
// ===== library: MasterCopy "Pulzer" =====

FUNCTION "Pulzer" : Void   // FC2, LAD
{ S7_Optimized_Access := 'FALSE' }
VERSION : 0.1
   VAR_INPUT
      T1 : Timer;
      T2 : Timer;
      Thigh : S5Time;
      Tdown : S5Time;
   END_VAR
   VAR_OUTPUT
      Q : Bool;
   END_VAR
   VAR_TEMP   // added for the SCL form of the ladder/FBD networks
      _w1 : Bool;
      _s5time1 : S5Time;
   END_VAR
BEGIN

REGION Network 1
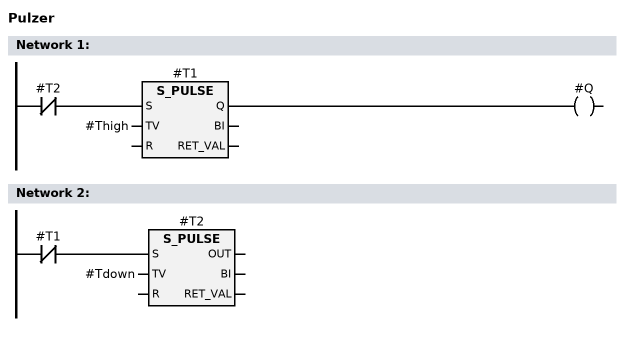
   RUNG wire#powerrail
      I_Contact( #T2 )
      S_PULSE(T_NO := #T1, TV := #Thigh, R :=, BI =>, RET_VAL =>)
      Coil( #Q )
   END_RUNG
   // the same network as SCL:
   #_s5time1 := S_PULSE(T_NO := #T1, S := NOT #T2, TV := #Thigh, Q => #_w1);
   #Q := #_w1;
END_REGION

REGION Network 2
   RUNG wire#powerrail
      I_Contact( #T1 )
      S_PULSE(T_NO := #T2, TV := #Tdown, R :=, BI =>, RET_VAL =>)
   END_RUNG
   // the same network as SCL:
   #_s5time1 := S_PULSE(T_NO := #T2, S := NOT #T1, TV := #Tdown);
END_REGION
END_FUNCTION

// ===== library: MasterCopy "Pallet dispenser" =====

FUNCTION_BLOCK "Pallet dispenser"   // FB4, LAD
{ S7_Optimized_Access := 'FALSE' }
VERSION : 0.1
   VAR_INPUT
      DOWN_accident : Bool;
      Dispenser_is_down : Bool;
      Dispenser_in_middle : Bool;
      Dispenser_is_up : Bool;
      UP_accident : Bool;
      Circuit_breaker : Bool;
      Arms_are_open : Bool;
      Arms_are_close : Bool;
      Pallet_under_dispenser : Bool;
      Automatic_mode : Bool;
      Power_circuit_OK : Bool;
      Pneumatic_OK : Bool;
      Sensor_before_dispenser : Bool;
      Button_Open_door : Bool;
      Sensor_door_are_open : Bool;
      Button_Door_are_close : Bool;
      OP_up : Bool;
      OP_down : Bool;
      OP_Airs_move : Bool;
      Pallet_transfare : Bool;
      Button_RESET : Bool;
      "Časovač 1" : Timer;
      "Časovač 2" : Timer;
      "Časovač 3" : Timer;
      "Časovač 4" : Timer;
      "Časovač 5" : Timer;
   END_VAR
   VAR_OUTPUT
      Let_go_UP : Bool;
      Let_go_DOWN : Bool;
      Break : Bool;
      Let_arms_close : Bool;
      Let_arms_open : Bool;
      Let_open_door : Bool;
      Led_door_are_open : Bool;
   END_VAR
   VAR
      Paleta_polozena : Bool;
      Stop_v_rucnim : Bool;
      Hrana_stop_v_rucnim : Bool;
      Pozadavek_otevreni_dveri : Bool;
      Door_opened : Bool;
      Arms_are_close_pozition : Bool;
   END_VAR
   VAR_TEMP   // added for the SCL form of the ladder/FBD networks
      _s5time1 : S5Time;
      _w1 : Bool;
   END_VAR
BEGIN

REGION Network 1
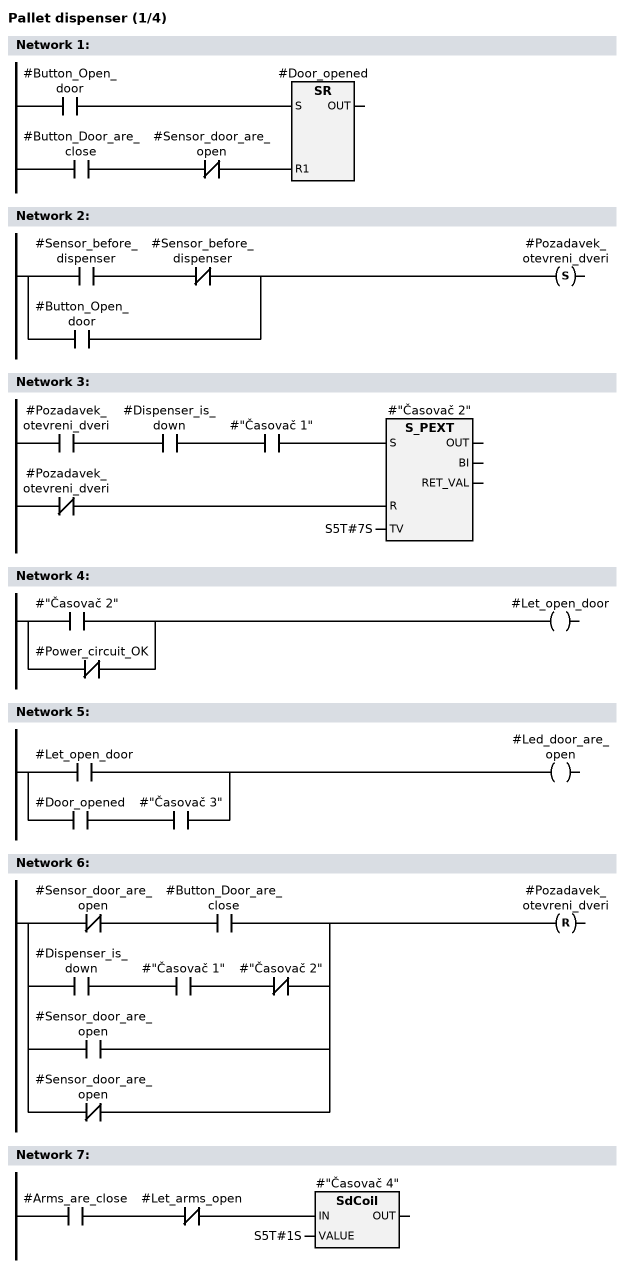
   RUNG wire#powerrail
      Contact( #Button_Open_door )
      S_SR(operand := #Door_opened, r1 := wire#w1)
   END_RUNG
   RUNG wire#powerrail
      Contact( #Button_Door_are_close )
      I_Contact( #Sensor_door_are_open )
   END_RUNG wire#w1
   // the same network as SCL:
   IF #Button_Open_door THEN
       #Door_opened := TRUE;   // SR flip-flop
   END_IF;
   IF #Button_Door_are_close AND NOT #Sensor_door_are_open THEN #Door_opened := FALSE; END_IF;
END_REGION

REGION Network 2
   RUNG wire#powerrail
      Contact( #Sensor_before_dispenser )
      I_Contact( #Sensor_before_dispenser )
      wire#w1
      S_Coil( #Pozadavek_otevreni_dveri )
   END_RUNG
   RUNG wire#powerrail
      Contact( #Button_Open_door )
   END_RUNG wire#w1
   // the same network as SCL:
   IF (#Sensor_before_dispenser AND NOT #Sensor_before_dispenser) OR #Button_Open_door THEN
       #Pozadavek_otevreni_dveri := TRUE;
   END_IF;
END_REGION

REGION Network 3
   RUNG wire#powerrail
      Contact( #Pozadavek_otevreni_dveri )
      Contact( #Dispenser_is_down )
      Contact( #"Časovač 1" )
      S_PEXT(T_NO := #"Časovač 2", R := wire#w1, TV := S5T#7S, BI =>, RET_VAL =>)
   END_RUNG
   RUNG wire#powerrail
      I_Contact( #Pozadavek_otevreni_dveri )
   END_RUNG wire#w1
   // the same network as SCL:
   #_s5time1 := S_PEXT(T_NO := #"Časovač 2",
                       S := #Pozadavek_otevreni_dveri AND #Dispenser_is_down AND #"Časovač 1",
                       R := NOT #Pozadavek_otevreni_dveri,
                       TV := S5T#7S);
END_REGION

REGION Network 4
   RUNG wire#powerrail
      Contact( #"Časovač 2" )
      wire#w1
      Coil( #Let_open_door )
   END_RUNG
   RUNG wire#powerrail
      I_Contact( #Power_circuit_OK )
   END_RUNG wire#w1
   // the same network as SCL:
   #Let_open_door := #"Časovač 2" OR NOT #Power_circuit_OK;
END_REGION

REGION Network 5
   RUNG wire#powerrail
      Contact( #Let_open_door )
      wire#w1
      Coil( #Led_door_are_open )
   END_RUNG
   RUNG wire#powerrail
      Contact( #Door_opened )
      Contact( #"Časovač 3" )
   END_RUNG wire#w1
   // the same network as SCL:
   #Led_door_are_open := #Let_open_door OR (#Door_opened AND #"Časovač 3");
END_REGION

REGION Network 6
   RUNG wire#powerrail
      I_Contact( #Sensor_door_are_open )
      Contact( #Button_Door_are_close )
      wire#w1
      R_Coil( #Pozadavek_otevreni_dveri )
   END_RUNG
   RUNG wire#powerrail
      Contact( #Dispenser_is_down )
      Contact( #"Časovač 1" )
      I_Contact( #"Časovač 2" )
   END_RUNG wire#w1
   RUNG wire#powerrail
      Contact( #Sensor_door_are_open )
   END_RUNG wire#w1
   RUNG wire#powerrail
      I_Contact( #Sensor_door_are_open )
   END_RUNG wire#w1
   // the same network as SCL:
   IF (NOT #Sensor_door_are_open AND #Button_Door_are_close) OR (#Dispenser_is_down AND #"Časovač 1" AND NOT #"Časovač 2") OR #Sensor_door_are_open OR NOT #Sensor_door_are_open THEN
       #Pozadavek_otevreni_dveri := FALSE;
   END_IF;
END_REGION

REGION Network 7
   // no SCL statement known for SdCoil: written as a call
   SdCoil(in := #Arms_are_close AND NOT #Let_arms_open, value := S5T#1S, operand := #"Časovač 4");
END_REGION

REGION Network 8
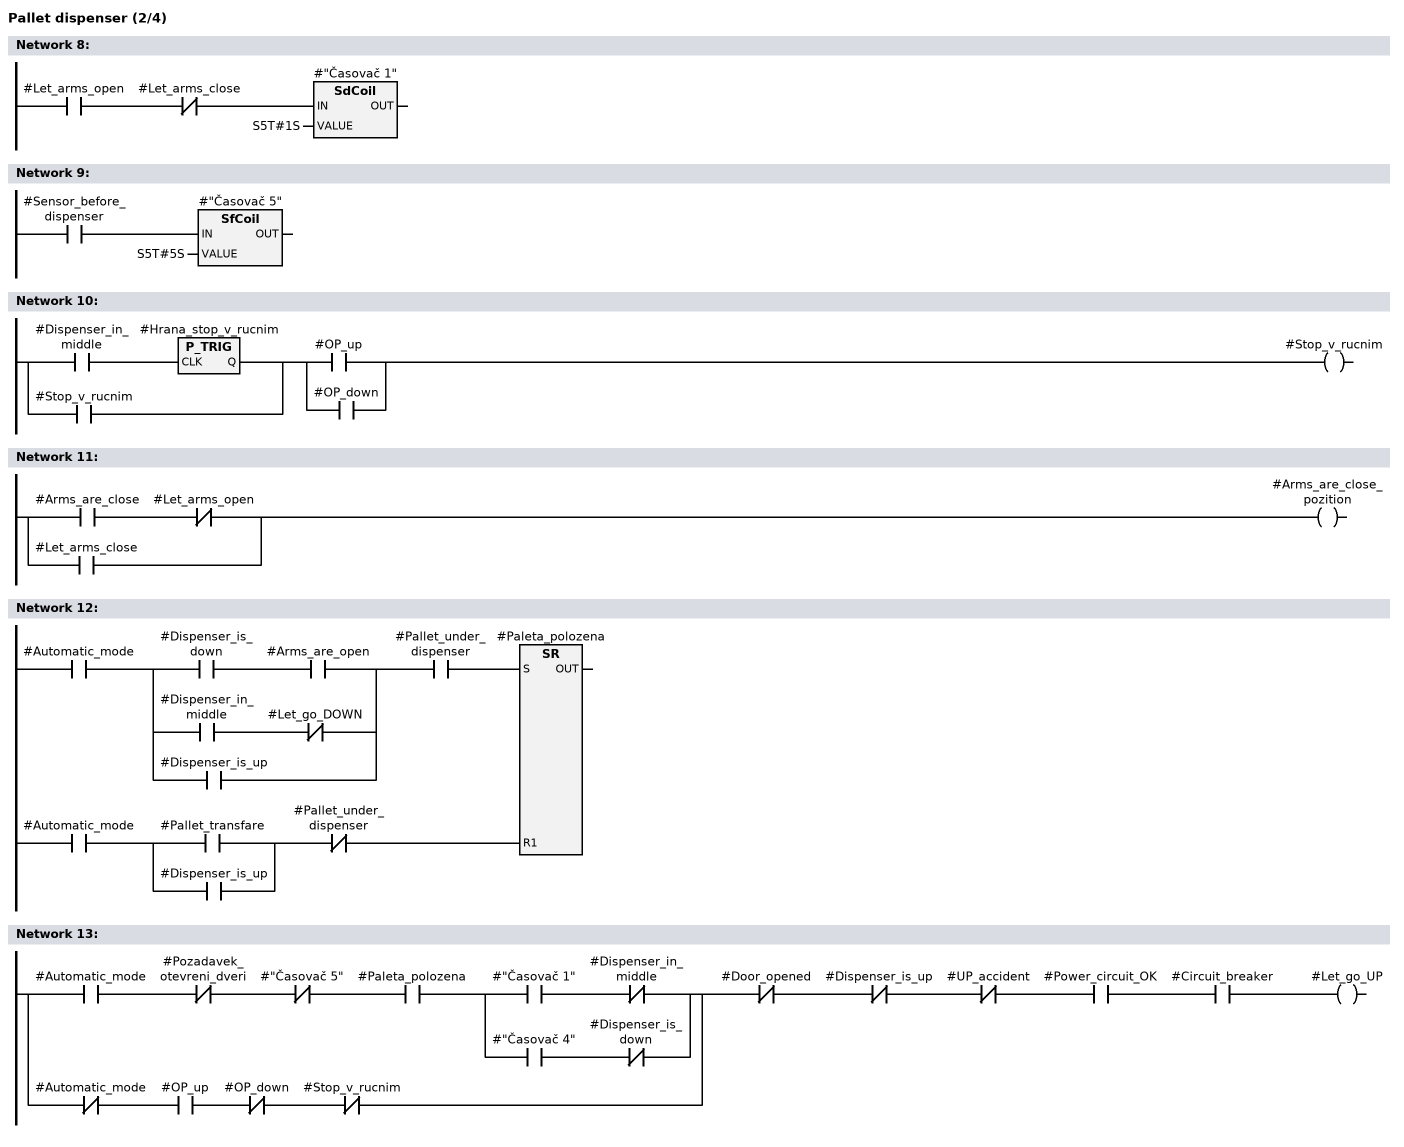
   // no SCL statement known for SdCoil: written as a call
   SdCoil(in := #Let_arms_open AND NOT #Let_arms_close, value := S5T#1S, operand := #"Časovač 1");
END_REGION

REGION Network 9
   // no SCL statement known for SfCoil: written as a call
   SfCoil(in := #Sensor_before_dispenser, value := S5T#5S, operand := #"Časovač 5");
END_REGION

REGION Network 10
   RUNG wire#powerrail
      Contact( #Dispenser_in_middle )
      P_Trig( #Hrana_stop_v_rucnim )
      wire#w1
      Contact( #OP_up )
      wire#w2
      Coil( #Stop_v_rucnim )
   END_RUNG
   RUNG wire#powerrail
      Contact( #Stop_v_rucnim )
   END_RUNG wire#w1
   RUNG wire#w1
      Contact( #OP_down )
   END_RUNG wire#w2
   // the same network as SCL:
   #_w1 := #Dispenser_in_middle AND NOT #Hrana_stop_v_rucnim;   // rising edge
   #Hrana_stop_v_rucnim := #Dispenser_in_middle;
   #Stop_v_rucnim := (#_w1 OR #Stop_v_rucnim) AND (#OP_up OR #OP_down);
END_REGION

REGION Network 11
   RUNG wire#powerrail
      Contact( #Arms_are_close )
      I_Contact( #Let_arms_open )
      wire#w1
      Coil( #Arms_are_close_pozition )
   END_RUNG
   RUNG wire#powerrail
      Contact( #Let_arms_close )
   END_RUNG wire#w1
   // the same network as SCL:
   #Arms_are_close_pozition := (#Arms_are_close AND NOT #Let_arms_open) OR #Let_arms_close;
END_REGION

REGION Network 12
   RUNG wire#powerrail
      Contact( #Automatic_mode )
      wire#w1
      Contact( #Dispenser_is_down )
      Contact( #Arms_are_open )
      wire#w2
      Contact( #Pallet_under_dispenser )
      S_SR(operand := #Paleta_polozena, r1 := wire#w5)
   END_RUNG
   RUNG wire#w1
      Contact( #Dispenser_in_middle )
      I_Contact( #Let_go_DOWN )
   END_RUNG wire#w2
   RUNG wire#w1
      Contact( #Dispenser_is_up )
   END_RUNG wire#w2
   RUNG wire#powerrail
      Contact( #Automatic_mode )
      wire#w3
      Contact( #Pallet_transfare )
      wire#w4
      I_Contact( #Pallet_under_dispenser )
   END_RUNG wire#w5
   RUNG wire#w3
      Contact( #Dispenser_is_up )
   END_RUNG wire#w4
   // the same network as SCL:
   IF #Automatic_mode AND ((#Dispenser_is_down AND #Arms_are_open) OR (#Dispenser_in_middle AND NOT #Let_go_DOWN) OR #Dispenser_is_up) AND #Pallet_under_dispenser THEN
       #Paleta_polozena := TRUE;   // SR flip-flop
   END_IF;
   IF #Automatic_mode AND (#Pallet_transfare OR #Dispenser_is_up) AND NOT #Pallet_under_dispenser THEN
       #Paleta_polozena := FALSE;
   END_IF;
END_REGION

REGION Network 13
   RUNG wire#powerrail
      Contact( #Automatic_mode )
      I_Contact( #Pozadavek_otevreni_dveri )
      I_Contact( #"Časovač 5" )
      Contact( #Paleta_polozena )
      wire#w1
      Contact( #"Časovač 1" )
      I_Contact( #Dispenser_in_middle )
      wire#w2
      I_Contact( #Door_opened )
      I_Contact( #Dispenser_is_up )
      I_Contact( #UP_accident )
      Contact( #Power_circuit_OK )
      Contact( #Circuit_breaker )
      Coil( #Let_go_UP )
   END_RUNG
   RUNG wire#w1
      Contact( #"Časovač 4" )
      I_Contact( #Dispenser_is_down )
   END_RUNG wire#w2
   RUNG wire#powerrail
      I_Contact( #Automatic_mode )
      Contact( #OP_up )
      I_Contact( #OP_down )
      I_Contact( #Stop_v_rucnim )
   END_RUNG wire#w2
   // the same network as SCL:
   #Let_go_UP := ((#Automatic_mode AND NOT #Pozadavek_otevreni_dveri AND NOT #"Časovač 5" AND #Paleta_polozena AND ((#"Časovač 1" AND NOT #Dispenser_in_middle) OR (#"Časovač 4" AND NOT #Dispenser_is_down))) OR (NOT #Automatic_mode AND #OP_up AND NOT #OP_down AND NOT #Stop_v_rucnim)) AND NOT #Door_opened AND NOT #Dispenser_is_up AND NOT #UP_accident AND #Power_circuit_OK AND #Circuit_breaker;
END_REGION

REGION Network 14
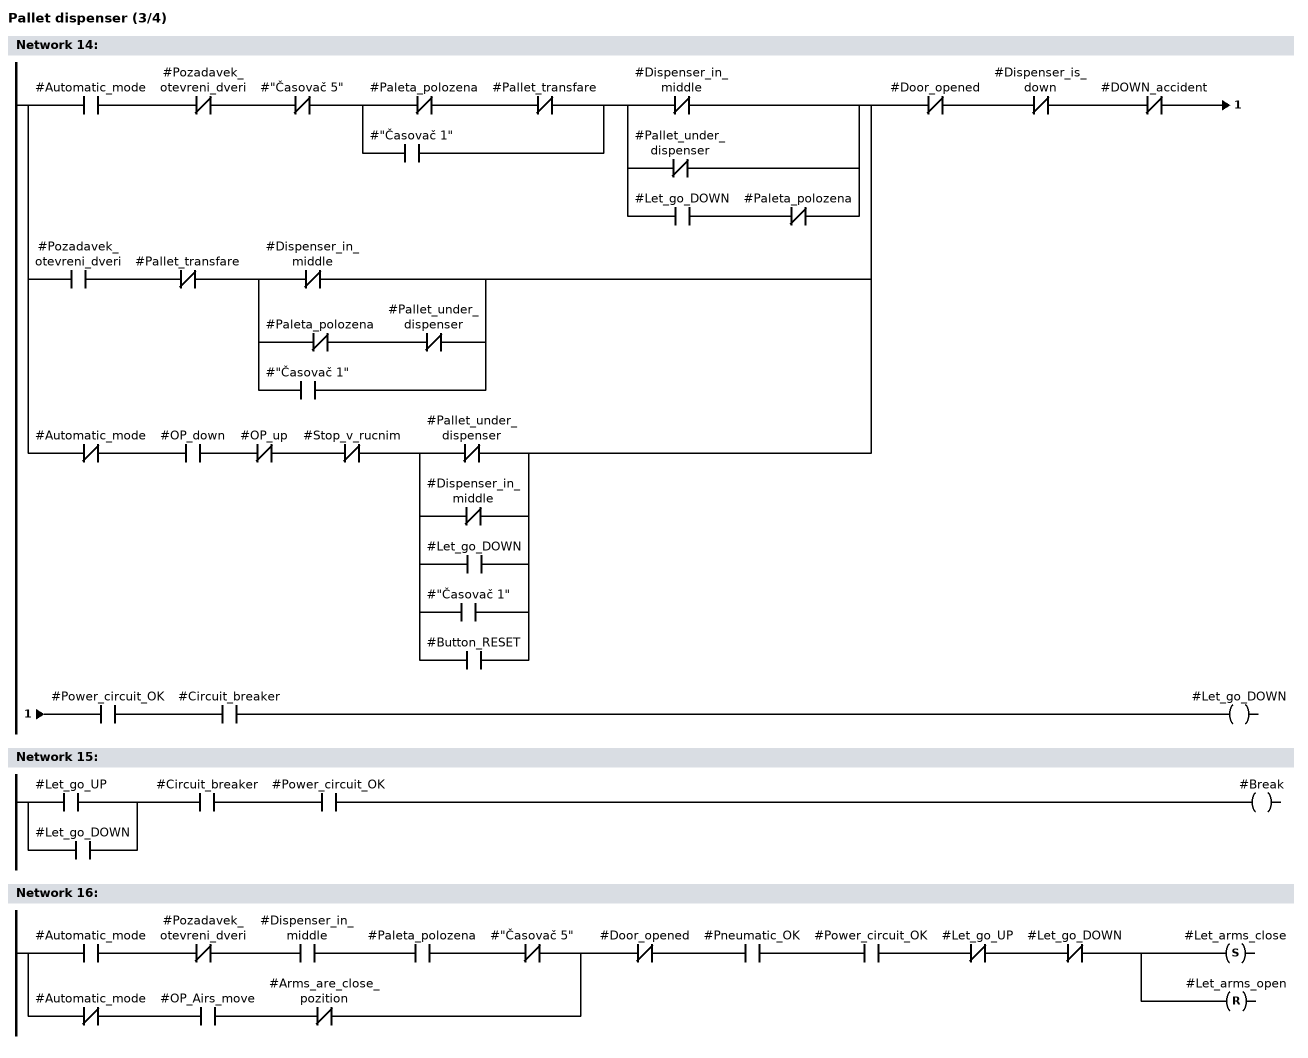
   RUNG wire#powerrail
      Contact( #Automatic_mode )
      I_Contact( #Pozadavek_otevreni_dveri )
      I_Contact( #"Časovač 5" )
      wire#w1
      I_Contact( #Paleta_polozena )
      I_Contact( #Pallet_transfare )
      wire#w2
      I_Contact( #Dispenser_in_middle )
      wire#w3
      I_Contact( #Door_opened )
      I_Contact( #Dispenser_is_down )
      I_Contact( #DOWN_accident )
      Contact( #Power_circuit_OK )
      Contact( #Circuit_breaker )
      Coil( #Let_go_DOWN )
   END_RUNG
   RUNG wire#w1
      Contact( #"Časovač 1" )
   END_RUNG wire#w2
   RUNG wire#w2
      I_Contact( #Pallet_under_dispenser )
   END_RUNG wire#w3
   RUNG wire#w2
      Contact( #Let_go_DOWN )
      I_Contact( #Paleta_polozena )
   END_RUNG wire#w3
   RUNG wire#powerrail
      Contact( #Pozadavek_otevreni_dveri )
      I_Contact( #Pallet_transfare )
      wire#w4
      I_Contact( #Dispenser_in_middle )
   END_RUNG wire#w3
   RUNG wire#w4
      I_Contact( #Paleta_polozena )
      I_Contact( #Pallet_under_dispenser )
   END_RUNG wire#w3
   RUNG wire#w4
      Contact( #"Časovač 1" )
   END_RUNG wire#w3
   RUNG wire#powerrail
      I_Contact( #Automatic_mode )
      Contact( #OP_down )
      I_Contact( #OP_up )
      I_Contact( #Stop_v_rucnim )
      wire#w5
      I_Contact( #Pallet_under_dispenser )
   END_RUNG wire#w3
   RUNG wire#w5
      I_Contact( #Dispenser_in_middle )
   END_RUNG wire#w3
   RUNG wire#w5
      Contact( #Let_go_DOWN )
   END_RUNG wire#w3
   RUNG wire#w5
      Contact( #"Časovač 1" )
   END_RUNG wire#w3
   RUNG wire#w5
      Contact( #Button_RESET )
   END_RUNG wire#w3
   // the same network as SCL:
   #Let_go_DOWN := ((#Automatic_mode AND NOT #Pozadavek_otevreni_dveri AND NOT #"Časovač 5" AND ((NOT #Paleta_polozena AND NOT #Pallet_transfare) OR #"Časovač 1") AND (NOT #Dispenser_in_middle OR NOT #Pallet_under_dispenser OR (#Let_go_DOWN AND NOT #Paleta_polozena))) OR (#Pozadavek_otevreni_dveri AND NOT #Pallet_transfare AND (NOT #Dispenser_in_middle OR (NOT #Paleta_polozena AND NOT #Pallet_under_dispenser) OR #"Časovač 1")) OR (NOT #Automatic_mode AND #OP_down AND NOT #OP_up AND NOT #Stop_v_rucnim AND (NOT #Pallet_under_dispenser OR NOT #Dispenser_in_middle OR #Let_go_DOWN OR #"Časovač 1" OR #Button_RESET))) AND NOT #Door_opened AND NOT #Dispenser_is_down AND NOT #DOWN_accident AND #Power_circuit_OK AND #Circuit_breaker;
END_REGION

REGION Network 15
   RUNG wire#powerrail
      Contact( #Let_go_UP )
      wire#w1
      Contact( #Circuit_breaker )
      Contact( #Power_circuit_OK )
      Coil( #Break )
   END_RUNG
   RUNG wire#powerrail
      Contact( #Let_go_DOWN )
   END_RUNG wire#w1
   // the same network as SCL:
   #Break := (#Let_go_UP OR #Let_go_DOWN) AND #Circuit_breaker AND #Power_circuit_OK;
END_REGION

REGION Network 16
   RUNG wire#powerrail
      Contact( #Automatic_mode )
      I_Contact( #Pozadavek_otevreni_dveri )
      Contact( #Dispenser_in_middle )
      Contact( #Paleta_polozena )
      I_Contact( #"Časovač 5" )
      wire#w1
      I_Contact( #Door_opened )
      Contact( #Pneumatic_OK )
      Contact( #Power_circuit_OK )
      I_Contact( #Let_go_UP )
      I_Contact( #Let_go_DOWN )
      wire#w2
      S_Coil( #Let_arms_close )
   END_RUNG
   RUNG wire#powerrail
      I_Contact( #Automatic_mode )
      Contact( #OP_Airs_move )
      I_Contact( #Arms_are_close_pozition )
   END_RUNG wire#w1
   RUNG wire#w2
      R_Coil( #Let_arms_open )
   END_RUNG
   // the same network as SCL:
   IF ((#Automatic_mode AND NOT #Pozadavek_otevreni_dveri AND #Dispenser_in_middle AND #Paleta_polozena AND NOT #"Časovač 5") OR (NOT #Automatic_mode AND #OP_Airs_move AND NOT #Arms_are_close_pozition)) AND NOT #Door_opened AND #Pneumatic_OK AND #Power_circuit_OK AND NOT #Let_go_UP AND NOT #Let_go_DOWN THEN
       #Let_arms_close := TRUE;
       #Let_arms_open := FALSE;
   END_IF;
END_REGION

REGION Network 17
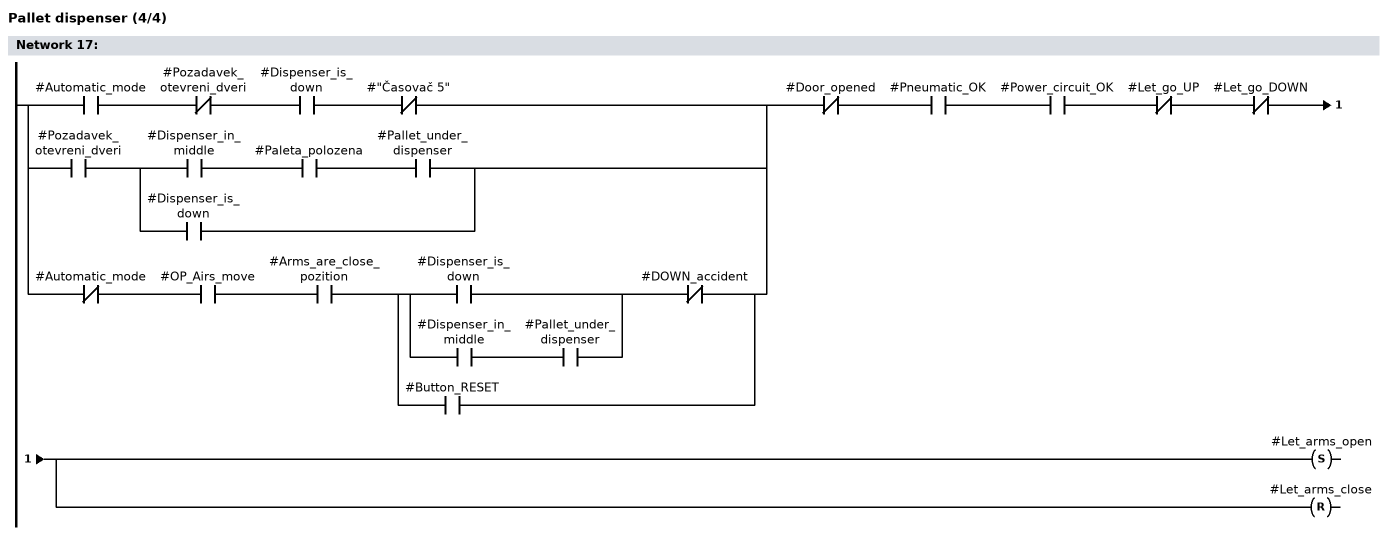
   RUNG wire#powerrail
      Contact( #Automatic_mode )
      I_Contact( #Pozadavek_otevreni_dveri )
      Contact( #Dispenser_is_down )
      I_Contact( #"Časovač 5" )
      wire#w1
      I_Contact( #Door_opened )
      Contact( #Pneumatic_OK )
      Contact( #Power_circuit_OK )
      I_Contact( #Let_go_UP )
      I_Contact( #Let_go_DOWN )
      wire#w5
      S_Coil( #Let_arms_open )
   END_RUNG
   RUNG wire#powerrail
      Contact( #Pozadavek_otevreni_dveri )
      wire#w2
      Contact( #Dispenser_in_middle )
      Contact( #Paleta_polozena )
      Contact( #Pallet_under_dispenser )
   END_RUNG wire#w1
   RUNG wire#w2
      Contact( #Dispenser_is_down )
   END_RUNG wire#w1
   RUNG wire#powerrail
      I_Contact( #Automatic_mode )
      Contact( #OP_Airs_move )
      Contact( #Arms_are_close_pozition )
      wire#w3
      Contact( #Dispenser_is_down )
      wire#w4
      I_Contact( #DOWN_accident )
   END_RUNG wire#w1
   RUNG wire#w3
      Contact( #Dispenser_in_middle )
      Contact( #Pallet_under_dispenser )
   END_RUNG wire#w4
   RUNG wire#w3
      Contact( #Button_RESET )
   END_RUNG wire#w1
   RUNG wire#w5
      R_Coil( #Let_arms_close )
   END_RUNG
   // the same network as SCL:
   IF ((#Automatic_mode AND NOT #Pozadavek_otevreni_dveri AND #Dispenser_is_down AND NOT #"Časovač 5") OR (#Pozadavek_otevreni_dveri AND ((#Dispenser_in_middle AND #Paleta_polozena AND #Pallet_under_dispenser) OR #Dispenser_is_down)) OR (NOT #Automatic_mode AND #OP_Airs_move AND #Arms_are_close_pozition AND (((#Dispenser_is_down OR (#Dispenser_in_middle AND #Pallet_under_dispenser)) AND NOT #DOWN_accident) OR #Button_RESET))) AND NOT #Door_opened AND #Pneumatic_OK AND #Power_circuit_OK AND NOT #Let_go_UP AND NOT #Let_go_DOWN THEN
       #Let_arms_open := TRUE;
       #Let_arms_close := FALSE;
   END_IF;
END_REGION
END_FUNCTION_BLOCK

// ===== library: MasterCopy "Vyhodnocení hran" =====

FUNCTION_BLOCK "Vyhodnocení hran"   // FB8, LAD
{ S7_Optimized_Access := 'FALSE' }
VERSION : 0.1
   VAR_INPUT
      input : DWord;
   END_VAR
   VAR_OUTPUT
      positive : DInt;
      negative : DInt;
   END_VAR
   VAR
      old_value : DWord;
   END_VAR
   VAR_TEMP
      change : DWord;
      invert : DWord;
   END_VAR
BEGIN

REGION Network 1
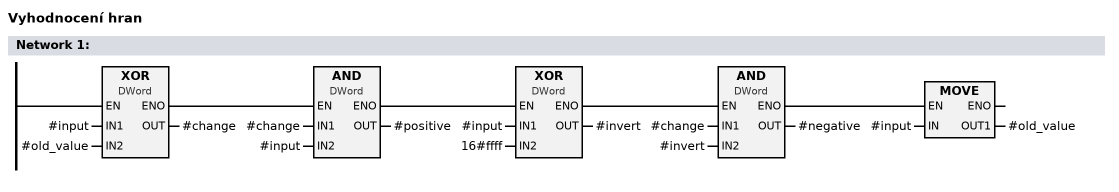
   // no checked SCL form for this network; see the picture
END_REGION
END_FUNCTION_BLOCK

// ===== library: MasterCopy "COMPLETE RESTART" =====

ORGANIZATION_BLOCK "COMPLETE RESTART"   // OB100, LAD
TITLE = "Complete Restart"
{ S7_Optimized_Access := 'FALSE' }
VERSION : 0.1
   VAR_TEMP
      OB100_EV_CLASS : Byte;   // 16#13, Event class 1, Entering event state, Event logged in diagnostic buffer
      OB100_STRTUP : Byte;   // 16#81/82/83/84 Method of startup
      OB100_PRIORITY : Byte;   // Priority of OB Execution
      OB100_OB_NUMBR : Byte;   // 100 (Organization block 100, OB100)
      OB100_RESERVED_1 : Byte;   // Reserved for system
      OB100_RESERVED_2 : Byte;   // Reserved for system
      OB100_STOP : Word;   // Event that caused CPU to stop (16#4xxx)
      OB100_STRT_INFO : DWord;   // Information on how system started
      OB100_DATE_TIME : Date_And_Time;   // Date and time OB100 started
   END_VAR
BEGIN

REGION Network 1
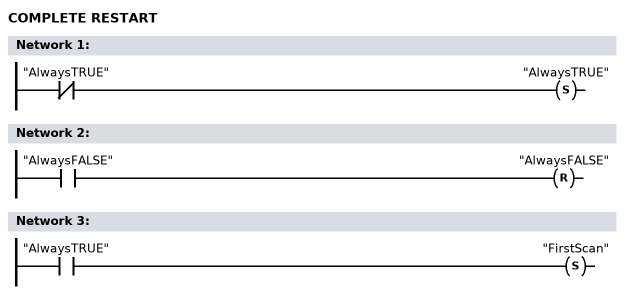
   RUNG wire#powerrail
      I_Contact( "AlwaysTRUE" )
      S_Coil( "AlwaysTRUE" )
   END_RUNG
   // the same network as SCL:
   IF NOT "AlwaysTRUE" THEN "AlwaysTRUE" := TRUE; END_IF;
END_REGION

REGION Network 2
   RUNG wire#powerrail
      Contact( "AlwaysFALSE" )
      R_Coil( "AlwaysFALSE" )
   END_RUNG
   // the same network as SCL:
   IF "AlwaysFALSE" THEN "AlwaysFALSE" := FALSE; END_IF;
END_REGION

REGION Network 3
   RUNG wire#powerrail
      Contact( "AlwaysTRUE" )
      S_Coil( "FirstScan" )
   END_RUNG
   // the same network as SCL:
   IF "AlwaysTRUE" THEN "FirstScan" := TRUE; END_IF;
END_REGION
END_ORGANIZATION_BLOCK